// Mitsubishi GX Works2 project: CydeusPlatform3   PLC: FX3U/FX3UC

TYPE ST_1SolCylinderInterface : STRUCT
  bBusy : BOOL;
  bError : BOOL;
  bDone : BOOL;
  bGoActive : BOOL;
  bReset : BOOL;
  tDelayTime : TIME;
  tTimeout : TIME;
END_STRUCT END_TYPE

TYPE ST_ServoMotorInterface : STRUCT
  bBusy : BOOL;
  bError : BOOL;
  bDone : BOOL;
  bServoEnabled : BOOL;
  bEnable : BOOL;
  bStop : BOOL;
  bAbort : BOOL;
  bReset : BOOL;
  bJogPos : BOOL;
  bJogNeg : BOOL;
  bMoveRel : BOOL;
  rMoveDist : REAL;
  iMoveVel : DINT;
  iMoveAccel : DINT;
END_STRUCT END_TYPE

// global labels: GVL_Error
VAR_GLOBAL
  arrError AT M200 : ARRAY [0..9] OF BOOL;
END_VAR
VAR_GLOBAL CONSTANT
  uiNumErrMinus1 : INT := 9;
END_VAR
VAR_GLOBAL
  arrMsg AT M250 : ARRAY [0..9] OF BOOL;
END_VAR
VAR_GLOBAL CONSTANT
  uiNumMsgMinus1 : INT := 9;
END_VAR

// global labels: GVL_Main
VAR_GLOBAL
  bAlarmTrigger : BOOL;
  bMachineError AT M100 : BOOL;
  bManualMode : BOOL;
  bAutoMode : BOOL;
  bStepMode : BOOL;
  bSimMode : BOOL;
  objPunching : CL_1Sol1SenCylinder;
  stServoMotor : ST_ServoMotorInterface;
  stPunching : ST_1SolCylinderInterface;
  objServoMotor : CL_ServoMotor;
  bManualEnable : BOOL;
  bMachineReady AT M101 : BOOL;
END_VAR

// global labels: GVL_HMI
VAR_GLOBAL
  btnInitialize AT M2 : BOOL;
  btnAutoMode AT M4 : BOOL;
  btnStepMode AT M5 : BOOL;
  btnTest AT M7 : BOOL;
  btnTestManualOn AT M8 : BOOL;
  btnSetup AT M9 : BOOL;
  btnStartAuto AT M11 : BOOL;
  tboxPulsePerRev AT D200 : DINT;
  tboxRadius AT D202 : REAL;
  tboxMoveVel AT D204 : DINT;
  tboxMoveAccel AT D206 : DINT;
  tboxPunchingDelayTime AT D210 : DINT;
  tboxPunchingTimeout AT D212 : DINT;
  btnServoStop AT M14 : BOOL;
  btnServoEnable AT M13 : BOOL;
  btnServoAbort AT M15 : BOOL;
  btnServoReset AT M16 : BOOL;
  btnServoJogPos AT M17 : BOOL;
  btnServoJogNeg AT M18 : BOOL;
  btnServoMoveRel AT M19 : BOOL;
  tboxMoveDist AT D126 : REAL;
  btnNextStep AT M6 : BOOL;
  btnStopAuto AT M12 : BOOL;
  btnLanguage AT D500 : INT;
  btnPunchingOutput AT M20 : BOOL;
  btnPunchingReset AT M21 : BOOL;
  btnManualMode AT M3 : BOOL;
  btnAbort AT M0 : BOOL;
  btnReset AT M1 : BOOL;
  btnBack AT M10 : BOOL;
  tboxProductLength AT D120 : INT;
  tboxNumProduct AT D121 : INT;
  btnRunContinuous AT M22 : BOOL;
  btnClearBatchCounter AT M23 : BOOL;
  tboxCycleTime AT D122 : REAL;
  btnManualOutput AT M24 : BOOL;
  btnMaPunchingOutput AT M25 : BOOL;
  btnMaServoPP AT M26 : BOOL;
  btnMaServoNP AT M27 : BOOL;
  btnMaServoEM2 AT M28 : BOOL;
  btnMaServoSON AT M29 : BOOL;
  btnMaServoRES AT M30 : BOOL;
  tboxCurrentProduct AT D130 : INT;
  btnInitialPunch AT M31 : BOOL;
  tboxRatio AT D214 : DINT;
END_VAR

// global labels: GVL_Output
VAR_GLOBAL
  boPunchingOutput AT Y006 : BOOL;
  bMaPunchingOutput : BOOL;
  bAuPunchingOutput : BOOL;
  boServoPP AT Y000 : BOOL;
  boServoNP AT Y001 : BOOL;
  boServoSON AT Y004 : BOOL;
  boServoRES AT Y005 : BOOL;
  boServoEM2 AT Y003 : BOOL;
  bMaServoPP : BOOL;
  bMaServoNP : BOOL;
  bMaServoSON : BOOL;
  bMaServoRES : BOOL;
  bMaServoEM2 : BOOL;
  bAuServoPP : BOOL;
  bAuServoNP : BOOL;
  bAuServoSON : BOOL;
  bAuServoRES : BOOL;
  bAuServoEM2 : BOOL;
END_VAR

// global labels: GVL_Input
VAR_GLOBAL
  biEstop1 AT X000 : BOOL;
  biEstop2 AT X001 : BOOL;
  biPunchingDone AT X002 : BOOL;
  biFeederSensor AT X003 : BOOL;
  biServoINP AT X005 : BOOL;
  biServoRD AT X006 : BOOL;
  biServoALM AT X007 : BOOL;
  bEstop1 : BOOL;
  bEstop2 : BOOL;
  bPunchingDone : BOOL;
  bFeederSensor : BOOL;
  bServoINP : BOOL;
  bServoRD : BOOL;
  bServoALM : BOOL;
END_VAR

// global labels: GVL_System
VAR_GLOBAL
  bCommandComplete AT M8029 : BOOL;
END_VAR

// global labels: GVL_StateMachine
VAR_GLOBAL
  bInitializingDone : BOOL;
  bInitializingAbort : BOOL;
  iStateInit : INT;
  iStateAuto AT D103 : INT;
  bAutoBatchDone : BOOL;
  bStopAutoHold : BOOL;
  bAbortDone : BOOL;
  iStateGeneral AT D100 : INT;
  iLastState AT D101 : INT;
  bResetBusy : BOOL;
  bAutoModeStarted AT M120 : BOOL;
  iStateTest AT D102 : INT;
  bManualModeReset : BOOL;
  iCurrentProduct : INT;
  tonCycleTime : TON;
  rCycleTime : REAL;
  tontemp : TON;
  btemp : BOOL;
END_VAR

// task Task_01 (event TRUE, interval 0, priority 31): MAIN

PROGRAM MAIN
VAR
  fbErrorController : FB_ErrorController;
  fbOutputController : FB_OutputController;
  fbStateMachine : FB_StateMachine;
  fbInputLinker : FB_InputLinker;
  fbObjectExecution : FB_ObjectExecution;
END_VAR

(*Input Linker*)
fbInputLinker();

(*State Machine*)
fbStateMachine();

(*Object Execution*)
fbObjectExecution();

(*Output Controller*)
fbOutputController();

(*Error Controller*)
fbErrorController(bResetError := btnReset);
bMachineError := fbErrorController.bError;
END_PROGRAM

FUNCTION_BLOCK FB_ErrorController
VAR
  ii : INT;
END_VAR
VAR_OUTPUT
  bError : BOOL;
END_VAR
VAR_INPUT
  bResetError : BOOL;
END_VAR
(*Error Controller*)

(*Reset Errors*)
IF bResetError THEN
	FOR ii := 0 TO uiNumErrMinus1  DO
		arrError[ii] := FALSE;
	END_FOR;
END_IF;

(*Register Errors*)
SET(bAlarmTrigger, arrError[0]);
SET(stPunching.bError, arrError[1]);
SET(stServoMotor.bError, arrError[2]);
SET(NOT bEstop1, arrError[3]);
SET(NOT bEstop2, arrError[4]);

(*Machine Error Trigger*)
bError := FALSE;
FOR ii := 0 TO uiNumErrMinus1  DO
	bError := bError OR arrError[ii];
END_FOR;

(*Register Messages*)
arrMsg[0] := NOT bFeederSensor;
arrMsg[1] := bAutoMode;
arrMsg[2] := bManualMode;
arrMsg[3] := bStepMode;
arrMsg[4] := btnTestManualOn;
arrMsg[5] := bMachineReady;
arrMsg[6] := bInitializingAbort;
END_FUNCTION_BLOCK

FUNCTION FUN_Output
VAR_INPUT
  b_OutAuto : BOOL;
  b_OutMan : BOOL;
  b_ManualMode : BOOL;
END_VAR
FUN_Output := (b_ManualMode AND b_OutMan) OR (NOT b_ManualMode AND b_OutAuto);
END_FUNCTION

FUNCTION_BLOCK FB_OutputController
(*Output Controller*)
(*Hold current status of output*)
IF LDP(TRUE, btnManualOutput) THEN
		btnMaPunchingOutput := boPunchingOutput ;
		btnMaServoEM2 := boServoEM2;
		btnMaServoNP := boServoNP;
		btnMaServoPP := boServoPP;
		btnMaServoRES := boServoRES;
		btnMaServoSON := boServoSON;
END_IF;

(*Calculate the logical output, then assign to physical output*)
boPunchingOutput := FUN_Output(btnManualOutput, bAuPunchingOutput, btnMaPunchingOutput);
boServoEM2:= FUN_Output(btnManualOutput, bAuServoEM2, btnMaServoEM2);
boServoNP:= FUN_Output(btnManualOutput, bAuServoNP, btnMaServoNP);
boServoPP:= FUN_Output(btnManualOutput, bAuServoPP, btnMaServoPP);
boServoRES:= FUN_Output(btnManualOutput, bAuServoRES, btnMaServoRES);
boServoSON:= FUN_Output(btnManualOutput, bAuServoSON, btnMaServoSON);
END_FUNCTION_BLOCK

FUNCTION_BLOCK FB_ManualMode
VAR
  arrTempHold : ARRAY [0..9] OF BOOL;
END_VAR
VAR CONSTANT
  iTempHoldSize : INT := 9;
END_VAR
VAR
  ii : INT;
END_VAR
(*Manual Mode*)
IF bManualModeReset THEN
		FOR ii := 0 TO iTempHoldSize DO 
			arrTempHold[ii] := FALSE;
		END_FOR;
END_IF;

IF (iStateGeneral = 60) OR (iStateGeneral = 100) THEN
		(*Enable Manual Mode*)
		bManualEnable := btnTestManualOn OR (iStateGeneral = 60);
		
		(*Hold Current status of Outputs*)
		IF LDP(TRUE, bManualEnable) THEN
			btnServoAbort := stServoMotor.bAbort;
			btnServoEnable := stServoMotor.bEnable;
			btnServoStop := stServoMotor.bStop;
			btnServoReset := stServoMotor.bReset OR btnReset;
			btnServoJogPos := stServoMotor.bJogPos;
			btnServoJogNeg := stServoMotor.bJogNeg;
			btnServoMoveRel := stServoMotor.bMoveRel;

			btnPunchingOutput := stPunching.bGoActive;
			btnPunchingReset := stPunching.bReset OR btnReset;
			
			arrTempHold[0] := stServoMotor.bAbort;
			arrTempHold[1] := stServoMotor.bEnable;
		END_IF;
		
		(*Restore status to output*)
		IF LDF(TRUE, bManualEnable ) THEN
			stServoMotor.bAbort := arrTempHold[0];
			stServoMotor.bEnable := arrTempHold[1];
		END_IF;
				
		(*Buttons on HMI control servo motor*)
		IF bManualEnable THEN
			stServoMotor.bAbort := btnServoAbort;
			stServoMotor.bEnable := btnServoEnable;
			stServoMotor.bStop := btnServoStop;
			stServoMotor.bReset := btnServoReset;
			stServoMotor.bJogPos := btnServoJogPos;
			stServoMotor.bJogNeg := btnServoJogNeg;
			stServoMotor.bMoveRel := btnServoMoveRel;
			stServoMotor.rMoveDist := tboxMoveDist;
			
			stPunching.bGoActive := btnPunchingOutput;
			stPunching.bReset := btnPunchingReset;
		END_IF;
END_IF;
END_FUNCTION_BLOCK

FUNCTION_BLOCK FB_Initializing
VAR
  fbDelayStep0 : TON;
  fbDelayStep10 : TON;
END_VAR
(*Initializing*)

IF iStateGeneral = 20 THEN
		(*State Machine*)
		CASE iStateInit OF
				0: 	(*Home the punching*)
						IF stPunching.bDone OR fbDelayStep0.Q THEN
								iStateInit := 10;
						END_IF;
						
				10:	(*Spare state*)
						IF (*stServoMotor.bServoEnabled*) TRUE THEN
								iStateInit := 20;
						ELSIF fbDelayStep10.Q THEN
								iStateInit := 50;
						END_IF;
						
				20: 	(*Done*)
						;
				50: 	(*Abort*)	
						;
		END_CASE;
		
		(*State Action*)
		RST((iStateInit = 0), stPunching.bGoActive);
		SET((iStateInit = 10), stServoMotor.bEnable);
		
		bInitializingDone := iStateInit = 20;
		bInitializingAbort := iStateInit = 50;				
END_IF;

(*Function block call*)
fbDelayStep0(IN := iStateInit = 0 AND NOT fbDelayStep0.Q, PT := t#2s);
fbDelayStep10(IN := iStateInit = 10 AND NOT fbDelayStep10.Q, PT := t#5s);
END_FUNCTION_BLOCK

FUNCTION_BLOCK FB_StateMachine
VAR
  fbInitializing : FB_Initializing;
  fbAutoMode : FB_AutoMode;
  fbManualMode : FB_ManualMode;
  fbAborting : FB_Aborting;
  fbReset : FB_Reset;
END_VAR
(*Main State Machine*)
IF (btnAbort OR bMachineError OR NOT bEstop1 OR NOT bEstop2) AND NOT (iStateGeneral = 10) AND NOT (iStateGeneral >= 100) THEN	(*Abort command*)
	iStateGeneral := 0;
END_IF;

IF btnReset  OR bResetBusy THEN
	fbReset();
END_IF;

CASE iStateGeneral OF
	0: 		(*Aborting*)
		IF bAbortDone THEN
			iStateGeneral := 10;
		END_IF;
	
	10: 		(*Begin*)
		IF btnInitialize AND NOT bMachineError THEN
			iStateGeneral := 20;
		ELSIF btnTest THEN
			iLastState := iStateGeneral;
			iStateGeneral := 100;
		ELSIF btnSetup THEN
			iLastState := iStateGeneral;
			iStateGeneral := 150;
		END_IF;
		
	20: 		(*Initializing*)
		IF bInitializingDone AND NOT bMachineError THEN
			iStateGeneral := 30;
		END_IF;
		
	30: 		(*Ready*)
		IF btnAutoMode AND NOT bMachineError THEN
			iStateGeneral := 40;
		ELSIF btnStepMode AND NOT bMachineError THEN
			iStateGeneral := 50;
		ELSIF btnManualMode AND NOT bMachineError THEN
			iStateGeneral := 60;
		ELSIF btnTest THEN
			iLastState := iStateGeneral;
			iStateGeneral := 100;
		END_IF;
	
	40: 		(*Running Auto Mode*)
		IF btnBack OR bAutoBatchDone  AND NOT bMachineError THEN
			iStateGeneral := 30;
		END_IF;
		
	50: 		(*Running Step Mode*)
		IF btnBack OR bAutoBatchDone AND NOT bMachineError THEN
			iStateGeneral := 30;
		END_IF;
		
	60: 		(*Running Manual Mode*)
		IF btnBack AND NOT bMachineError THEN
			iStateGeneral := 30;
		END_IF;
		
	100: 		(*Testing*)
		IF btnBack THEN
			iStateGeneral := iLastState;
		END_IF;
		
	150: 		(*Setting*)
		IF btnBack THEN
			iStateGeneral := iLastState;
		END_IF;
	
ELSE 
		;
END_CASE;

(*State Action*)
bAutoMode := iStateGeneral = 40;
bStepMode := iStateGeneral = 50;
bManualMode := iStateGeneral = 60;
bMachineReady := (iStateGeneral >= 30) AND (iStateGeneral < 100);
IF LDP(TRUE, iStateGeneral = 100) THEN
		iStateTest := 0;
END_IF;	

stServoMotor.bEnable := (iStateGeneral >= 40) AND (iStateGeneral <= 60);

		(*Clear product counter*)
		IF btnClearBatchCounter THEN
				iCurrentProduct := 0;
				tboxCurrentProduct := 0;
				tboxCycleTime := 0.0;
		END_IF;

(*Function Block Call*)
bInitializingDone := FALSE;
bInitializingAbort := FALSE;
bAutoBatchDone := FALSE;
bAbortDone := FALSE;
bAutoModeStarted := FALSE;

fbAborting();
fbInitializing();
fbAutoMode(bEnStepMode := iStateGeneral = 50, bNext := btnNextStep);
fbManualMode();
END_FUNCTION_BLOCK

FUNCTION_BLOCK FB_AutoMode
VAR_INPUT
  bEnStepMode : BOOL;
END_VAR
VAR
  bState80 : BOOL;
END_VAR
VAR_INPUT
  bNext : BOOL;
END_VAR
VAR
  bNextStep : BOOL;
  bExit : BOOL;
  bDelayState : BOOL;
END_VAR
(*Initialize and Reset Function Block*)

IF iStateGeneral = 40 OR iStateGeneral = 50 THEN
		(*Auto Mode State Machine*)
		CASE iStateAuto OF
				0: 		(*Ready*)
						IF btnStartAuto THEN
							iStateAuto := 10;
						END_IF;
						
				10: 		(*Wait for raw material*)
						IF bFeederSensor AND bNextStep THEN
							iStateAuto := 15;
						END_IF;
						
				15:		(*Check if Initial punch needed*)
						IF btnInitialPunch THEN
							iStateAuto := 20;
						ELSE
							iStateAuto := 30;
						END_IF;
						
				20: 		(*Cut spare material before beginning*)
						IF stPunching.bDone AND bNextStep THEN
							iStateAuto := 30;
						END_IF;
						
				30: 		(*Set parameters*)
						bDelayState := NOT bDelayState;
						stServoMotor.rMoveDist := INT_TO_REAL(tboxProductLength);
						IF bDelayState THEN
							iStateAuto := 40;
						END_IF;
				
				40: 		(*Feed new raw material to punching machine*)
						IF stServoMotor.bDone AND bNextStep THEN
							iStateAuto := 50;
						END_IF;
					
				50: 		(*Cut raw material into final product*)
						IF stPunching.bDone AND bNextStep THEN
							iStateAuto := 60;
						END_IF;
						
				60: 		(*Count a completed product*)
						iCurrentProduct := iCurrentProduct + 1;
						iStateAuto := 70;
		
				70: 		(*Check for raw material*)
						IF (NOT bFeederSensor OR (iCurrentProduct >= tboxNumProduct AND NOT btnRunContinuous)) AND NOT bStopAutoHold THEN
							iStateAuto := 80;
						ELSIF bFeederSensor AND NOT bStopAutoHold THEN
							iStateAuto := 30;
						ELSIF bStopAutoHold THEN 
							iStateAuto := 100;
						END_IF;
						
				80: 		(*Auto mode done*)
						;
						
				100: 	(*Stop*)
						IF btnStartAuto THEN
							iStateAuto := 30;
						ELSIF bExit THEN 
							iStateAuto := 80;
						END_IF;
						
		END_CASE;
		
		(*Auto Mode State Action*)
		bNextStep := (NOT bEnStepMode OR (bEnStepMode AND bNext));
		SET(btnStopAuto, bStopAutoHold);
		RST(iStateAuto = 100, bStopAutoHold);
		bAutoBatchDone:= iStateAuto = 80;
		bAutoModeStarted := iStateAuto >= 10 AND iStateAuto < 100;
		
		stServoMotor.bMoveRel := (iStateAuto = 40);
		stPunching.bGoActive := (iStateAuto = 20) OR (iStateAuto = 50);
		
ELSIF iStateGeneral = 30 THEN
		iStateAuto := 0;
		bStopAutoHold := FALSE;
END_IF;

(*Cycle time calculation*)
IF (iStateAuto = 60) OR  (iStateAuto = 70) THEN
		tboxCycleTime := rCycleTime;
		tboxCurrentProduct := iCurrentProduct;
END_IF;

IF iStateAuto = 30 THEN
		rCycleTime := 0.0;
END_IF;

tonCycleTime(IN := NOT tonCycleTime.Q AND ((iStateAuto = 40) OR (iStateAuto = 50)), PT := t#100ms);
IF tonCycleTime.Q THEN
		rCycleTime := rCycleTime + 0.1;
END_IF;
END_FUNCTION_BLOCK

FUNCTION_BLOCK FB_InputLinker
(*Input Linker*)

(*Link physical input to logical input memory*)
IF NOT bSimMode THEN	
		bEstop1 := biEstop1;
		bEstop2 := biEstop2;
		bFeederSensor := biFeederSensor;
		bPunchingDone := biPunchingDone;
		bServoINP := biServoINP;
		bServoRD := biServoRD;
		bServoALM := biServoALM;
END_IF;
END_FUNCTION_BLOCK

FUNCTION_BLOCK FB_ObjectExecution
objServoMotor(biINP := bServoINP,
								biRD := bServoRD,
								biALM := bServoALM,
								boNPz := bAuServoNP,
								boEM2 := bAuServoEM2,
								boRES := bAuServoRES,
								boSON := bAuServoSON,
								
								bEnable := stServoMotor.bEnable,
								bStop := stServoMotor.bStop,
								bAbort := stServoMotor.bAbort,
								bReset := stServoMotor.bReset,
								iOutChannel := 0,
								iRevChannel := 1,
								iMoveDelay := 100,
								iPulsePerRev := tboxPulsePerRev,
								rRadius := tboxRadius,
								iRatio := tboxRatio,
								
								bJogPos := stServoMotor.bJogPos,
								bJogNeg := stServoMotor.bJogNeg,
								
								bMoveRel := stServoMotor.bMoveRel,
								rMoveDist := stServoMotor.rMoveDist,
								iMoveVel := (tboxMoveVel*tboxRatio),
								iMoveAccel := tboxMoveAccel,

								bBusy := stServoMotor.bBusy,
								bDone := stServoMotor.bDone,
								bError := stServoMotor.bError,
								bServoEnabled := stServoMotor.bServoEnabled);
								
								
objPunching(biSensorDone := bPunchingDone,
							biActiveFeedback := bAuPunchingOutput,
							boSolenoid := bAuPunchingOutput,
							
							bGoActive := stPunching.bGoActive,
							bReset := stPunching.bReset,
							tDelayTime := tboxPunchingDelayTime,
							tTimeout := tboxPunchingTimeout,

							bBusy := stPunching.bBusy,
							bDone := stPunching.bDone,
							bError := stPunching.bError);
END_FUNCTION_BLOCK

FUNCTION_BLOCK CL_1Sol1SenCylinder
VAR_INPUT
  biSensorDone : BOOL;
  bGoActive : BOOL;
  bReset : BOOL;
END_VAR
VAR_OUTPUT
  boSolenoid : BOOL;
  bBusy : BOOL;
  bInHomePos : BOOL;
  bError : BOOL;
END_VAR
VAR_INPUT
  tDelayTime : DINT;
  tTimeout : DINT;
END_VAR
VAR
  fbDelayTime : TON;
  fbTimeout : TON;
END_VAR
VAR_INPUT
  biActiveFeedback : BOOL;
END_VAR
VAR
  bSensorDoneHold : BOOL;
  tDelay : TIME;
  tTimeoutz : TIME;
END_VAR
VAR_OUTPUT
  bDone : BOOL;
END_VAR
(*Activate Output: Enable solenoid on valve*) 
boSolenoid := LDP(TRUE, bGoActive) OR boSolenoid AND NOT fbTimeout.Q AND NOT biSensorDone;

(*Process Input: Wait for sensors signal*)
SET(biSensorDone, bSensorDoneHold);
RST(LDP(TRUE, bBusy), bSensorDoneHold);
bInHomePos := fbDelayTime.Q AND bSensorDoneHold;
bBusy := biActiveFeedback AND NOT biSensorDone;
bDone := NOT bBusy AND bGoActive;

(*Error handling*)
		(*Notify timeout error*)
		SET(fbTimeout.Q, bError);

		(*Reset timeout error*)
		RST(bReset, bError);

(*Timers call*)
tDelay := DINT_TO_TIME(tDelayTime);
tTimeoutz := DINT_TO_TIME(tTimeout);
fbDelayTime(IN := NOT bBusy, PT := tDelay );
fbTimeout(IN := bBusy, PT := tTimeoutz );
END_FUNCTION_BLOCK

FUNCTION_BLOCK FB_Aborting
VAR
  fbAbortHold : TP;
  ini : INT;
  outi : INT;
END_VAR
(*Aborting*)

IF iStateGeneral = 0 THEN
		(*Abort object*)
		stServoMotor.bEnable := FALSE;
		stServoMotor.bAbort := fbAbortHold.Q;
		stServoMotor.bStop := FALSE;
		stServoMotor.bJogNeg := FALSE;
		stServoMotor.bJogPos := FALSE;
		stServoMotor.bMoveRel := FALSE;
		
		stPunching.bGoActive := FALSE;
		
		(*About function block*)
		bManualModeReset := fbAbortHold.Q;
		
		(*Clear variables*)
		iStateInit := 0;
		iStateAuto := 0;
		bStopAutoHold := FALSE;
		iCurrentProduct := 0;
		rCycleTime := 0.0;
		
		bAbortDone := NOT btnAbort AND NOT fbAbortHold.Q;
END_IF;

fbAbortHold(IN := btnAbort OR fbAbortHold.Q, PT := t#1000ms);
END_FUNCTION_BLOCK

FUNCTION_BLOCK FB_Reset
stPunching.bReset := btnReset;
stServoMotor.bReset := btnReset;
bResetBusy := btnReset;
END_FUNCTION_BLOCK

FUNCTION_BLOCK CL_ServoMotor
VAR_INPUT
  biINP : BOOL;
  biRD : BOOL;
  biALM : BOOL;
  bEnable : BOOL;
  bStop : BOOL;
  bAbort : BOOL;
  bReset : BOOL;
  bJogPos : BOOL;
  bJogNeg : BOOL;
  bMoveRel : BOOL;
  rMoveDist : REAL;
END_VAR
VAR_OUTPUT
  boEM2 : BOOL;
  boSON : BOOL;
  boRES : BOOL;
  bBusy : BOOL;
  bError : BOOL;
  bDone : BOOL;
  bServoEnabled : BOOL;
END_VAR
VAR
  iState : INT;
  fbResetHold : TP_10;
  bResetHold : BOOL;
  fbMoveDelay : TON;
END_VAR
VAR_INPUT
  iMoveDelay : WORD;
END_VAR
VAR
  tMoveDelay : TIME;
  iStopState : INT;
END_VAR
VAR_INPUT
  iMoveVel : DINT;
  iMoveAccel : DINT;
  iPulsePerRev : DINT;
  rRadius : REAL;
END_VAR
VAR
  iFrequency : DINT;
  iPulse : DINT;
  iAccel : DINT;
  bOutPulse : BOOL;
END_VAR
VAR_INPUT
  iOutChannel : INT;
  iRevChannel : INT;
END_VAR
VAR
  bInCommand : BOOL;
  bCompleted : BOOL;
  tonDelayComplete : TON_10;
  bCompletedHold : BOOL;
  bDebug : BOOL;
END_VAR
VAR_OUTPUT
  boNPz : BOOL;
END_VAR
VAR_INPUT
  iRatio : DINT;
END_VAR
(*Main State Machine*)
CASE iState OF 
		0: 	(*Unenabled, wait for Enable command*)
				IF bEnable AND NOT bStop AND NOT bError THEN
						iState := 10;
				END_IF;
				
		10: 	(*Servo On*)
				IF bServoEnabled THEN
						iState := 20;
				END_IF;
						
		20: 	(*Servo Ready, wait for moving command*)
				IF bJogPos AND NOT bStop AND NOT bError THEN
						iState := 100;
				ELSIF bJogNeg AND NOT bStop AND NOT bError THEN
						iState := 140;
				ELSIF bMoveRel AND NOT bStop AND NOT bError THEN
						iState := 200;
				END_IF;
				
		100: 	(*Calculate number of pulse*)			
				iFrequency := 2000;
				iPulse := REAL_TO_DINT(DINT_TO_REAL(iRatio*iPulsePerRev)*1000.0/(2.0*3.1415926*rRadius));
				iAccel := iMoveAccel;
				iState := 110;
				
		110: 	(*Execute Jog Pos command*)
				IF NOT bJogPos THEN 
						iState := 20;
				END_IF;
				
		140: 	(*Calculate number of pulse*)			
				iFrequency := 2000;
				iPulse := REAL_TO_DINT(DINT_TO_REAL(iRatio*iPulsePerRev)*1000.0/(2.0*3.1415926*rRadius));
				iAccel := iMoveAccel;
				iState := 150;
				
		150: 	(*Execute Jog Neg command*)
				IF NOT bJogNeg THEN
						iState := 20;
				END_IF;
				
		200: 	(*Calculate number of pulse*)
				iFrequency := REAL_TO_DINT(DINT_TO_REAL(iPulsePerRev*iMoveVel)/60.0);
				iPulse := REAL_TO_DINT(DINT_TO_REAL(iRatio*iPulsePerRev)*rMoveDist/(2.0*3.1415926*rRadius));	
				iAccel := iMoveAccel;
				tMoveDelay := WORD_TO_TIME(iMoveDelay);
				iState := 210;
		
		210: 	(*Execute Move Relative command*)
				IF tonDelayComplete.Q AND fbMoveDelay.Q THEN		
						iState := 220;
				END_IF;		
				
		220: 	(*Move Relative done, wait for command release*)
				IF NOT bMoveRel THEN
						iState := 20;
				END_IF;
				
END_CASE;
	
(*Procedure*)
		(*Abort*)
		IF bAbort OR NOT bEnable OR bError THEN
				iState := 0;
				iStopState := 0;
		END_IF;
		
		(*Reset*)
		IF bReset AND bError THEN
				iState := 0;
				iStopState := 0;
		END_IF;		
		
		(*Stop*)
		CASE iStopState OF
				0: 	(*Wait for stop signal*)
						IF bStop THEN
								iStopState := 10;
						END_IF;
						
				10: 	(*Execute Stop*)
						IF iState > 20 THEN
								iState := 20;
						END_IF;
						IF biINP THEN
								iStopState := 20;
						END_IF;
						
				20: 	(*Stop done, wait for command release*)
						IF NOT bStop THEN
								iStopState := 0;
						END_IF;
		END_CASE;	

(*State Action*)
		boSON := (iState >= 10);																			(*Enable Servo Motor*)	
		boEM2 := NOT bAbort AND biALM;													(*Abort Servo Motor*)
		boRES := fbResetHold.Q AND NOT biALM;									(*Reset Servo Motor*)		
		
		bBusy := (iState = 110) OR (iState = 150) OR (iState = 210) OR (iStopState = 10);
		bDone := (iState = 220) OR (iStopState = 20);									(*Servo movement is done*)
		bServoEnabled := biRD;																		(*Servo is powered on*)
	
		SET(NOT biALM, bError);																		(*Notify Servo Motor Error*)
		RST((bReset AND bError), bError);													(*Reset object error*)	
		
		bInCommand:= ((iState = 110) OR (iState = 150) OR (iState = 210)) AND NOT (iStopState = 10);	(*Enable Pulse*)
		boNPz := ((iState = 150) OR (rMoveDist < 0.0));												(*Reverse rotation*)
		
		SET(bCompleted, bCompletedHold);
		RST(NOT (iState = 210), bCompletedHold);
		bResetHold := (bReset AND NOT fbResetHold.Q) OR (bResetHold AND fbResetHold.Q) ;
	
(*Function Block Call*)
fbResetHold(IN := bResetHold, PT := t#600ms);
fbMoveDelay(IN := (iState = 210) AND bServoEnabled AND NOT bStop AND NOT bAbort AND NOT bError, PT := tMoveDelay);
tonDelayComplete(IN := biINP AND bCompletedHold, PT:= t#50ms);

(*Output pulse to server drive*)
bOutPulse := (LDP(TRUE, bInCommand) OR bOutPulse) AND NOT (bCompleted AND bMoveRel) AND NOT LDF(TRUE, bInCommand);		(*Output pulse command*)

CASE iOutChannel OF 
	0: 	(*Y000*)
			DPLSR(bOutPulse, iFrequency, iPulse, iAccel, Y000);
			bDebug := M8013;
	1:		(*Y001*)
			DPLSR(bOutPulse, iFrequency, iPulse, iAccel, Y001);
	2:		(*Y002*)
			DPLSR(bOutPulse, iFrequency, iPulse, iAccel, Y002);
END_CASE;
bCompleted := bCommandComplete;
END_FUNCTION_BLOCK
